Fanuc KAREL source: KO00137.KL

PROGRAM KO00137
%NOLOCKGROUP
VAR
  R: REAL
  CFG: CONFIG
  OUT: XYZWPR
  N: INTEGER
BEGIN
  N = 1
  R = 2.0
  CFG.CFG_FLIP = TRUE
  OUT = POS(R, R, N, R, R, R, CFG)
END KO00137
